// TIA Portal project "bai5" (V15)

(* hardware
DEVICE "S7-1200 station_1"  S7-1200 Station
   slot 0: "Rack_0"  S7-1200 Rack  Rack  V1.0
   slot 1: "PLC_1"  CPU 1214C DC/DC/Rly  6ES7 214-1HG40-0XB0  V4.2
*)

// ===== PLC "PLC_1"  CPU 1214C DC/DC/Rly =====

VAR_GLOBAL   // PLC tag table "Default tag table"
   "start" AT %M2.0 : Bool;
   "stop" AT %M2.1 : Bool;
   "quaynguoc" AT %Q0.0 : Bool;
   "nutthuan" AT %M2.2 : Bool;
   "quaythuan" AT %Q0.1 : Bool;
   "nutnguoc" AT %M2.3 : Bool;
END_VAR

// folder: System blocks/Program resources

DATA_BLOCK "IEC_Timer_0_DB"   // DB1
{ S7_Optimized_Access := 'TRUE' }
AUTHOR : Simatic
FAMILY : IEC
NAME : IEC_TMR
VERSION : 1.0
// stored: InstanceOfName IEC_TIMER
"IEC_TIMER"
BEGIN
END_DATA_BLOCK

DATA_BLOCK "IEC_Timer_0_DB_1"   // DB2
{ S7_Optimized_Access := 'TRUE' }
AUTHOR : Simatic
FAMILY : IEC
NAME : IEC_TMR
VERSION : 1.0
// stored: InstanceOfName IEC_TIMER
"IEC_TIMER"
BEGIN
END_DATA_BLOCK

DATA_BLOCK "IEC_Timer_0_DB_2"   // DB3
{ S7_Optimized_Access := 'TRUE' }
AUTHOR : Simatic
FAMILY : IEC
NAME : IEC_TMR
VERSION : 1.0
// stored: InstanceOfName IEC_TIMER
"IEC_TIMER"
BEGIN
END_DATA_BLOCK

// folder: (top level)

ORGANIZATION_BLOCK "Main"   // OB1, LAD, ProgramCycle
TITLE = "Main Program Sweep (Cycle)"
{ S7_Optimized_Access := 'TRUE' }
VERSION : 0.1
   VAR_INPUT
      Initial_Call : Bool;   // Initial call of this OB
      Remanence : Bool;   // =True, if remanent data are available
   END_VAR
BEGIN

REGION Network 1
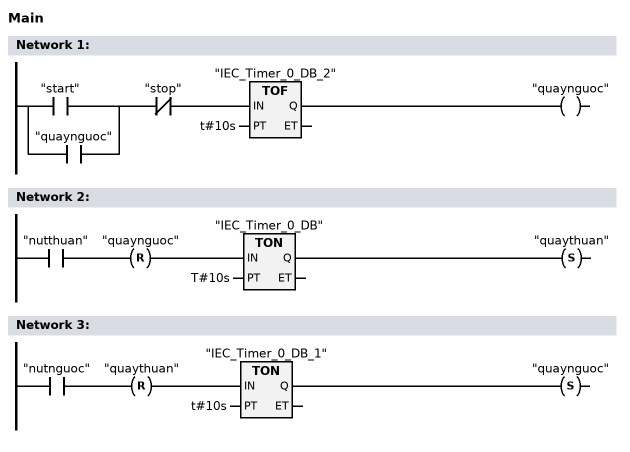
   "IEC_Timer_0_DB_2".TOF(IN := ("start" OR "quaynguoc") AND NOT "stop", PT := t#10s);
   "quaynguoc" := "IEC_Timer_0_DB_2".Q;
END_REGION

REGION Network 2
   IF "nutthuan" THEN "quaynguoc" := FALSE; END_IF;
   "IEC_Timer_0_DB".TON(IN := "nutthuan", PT := T#10s);
   IF "IEC_Timer_0_DB".Q THEN "quaythuan" := TRUE; END_IF;
END_REGION

REGION Network 3
   IF "nutnguoc" THEN "quaythuan" := FALSE; END_IF;
   "IEC_Timer_0_DB_1".TON(IN := "nutnguoc", PT := t#10s);
   IF "IEC_Timer_0_DB_1".Q THEN "quaynguoc" := TRUE; END_IF;
END_REGION
END_ORGANIZATION_BLOCK